// TIA Portal V20 export
DATA_BLOCK "HmiInterface"   // DB141
// stored: Access Published, MemoryReserve 100, Namespace Unit1.Em0
   VAR
      em : "LAF_typeEmInterface";
      stacker1NgBox : "LER_typeSequenceInterface";
      cmStacker1NgBoxDetect : "LBC_typeDigitalSignalInterface";
      cmStacker1NgBoxFullDetect : "LBC_typeDigitalSignalInterface";
      cmStacker1NgBoxLoadingUpDown : "LBC_typeTwoWayActuatorInterface";
      cmStacker1NgBoxUnitMoverBwdFwd : "LBC_typeTwoWayActuatorInterface";
      cmStacker1NgBoxClampLeftOpenClose : "LBC_typeTwoWayActuatorInterface";
      cmStacker1NgBoxClampRightOpenClose : "LBC_typeTwoWayActuatorInterface";
      cmStacker1NgBoxClampMoverOpenClose : "LBC_typeTwoWayActuatorInterface";
      cmStacker1NgBoxLiftDownUp : "LBC_typeTwoWayActuatorInterface";
      cmStacker1NgBoxLockDownUp : "LBC_typeTwoWayActuatorInterface";
      intCondition : "Unit1.Em0.typeIntConditionHmiInterface";
   END_VAR
BEGIN
   cmStacker1NgBoxLoadingUpDown.configuration.referenceDesignator := WSTRING#'STAKC #1 NG CLAMP Z-AXIS';
   cmStacker1NgBoxClampLeftOpenClose.configuration.referenceDesignator := WSTRING#'STACK #1 NG CLAMP LEFT';
   cmStacker1NgBoxClampRightOpenClose.configuration.referenceDesignator := WSTRING#'STACK #1 NG CLAMP RIGHT';
   cmStacker1NgBoxClampMoverOpenClose.configuration.referenceDesignator := WSTRING#'STACK #1 NG CLAMP MOVER';
END_DATA_BLOCK
